FUNCTION_BLOCK Test_DateTimeAsString_ms EXTENDS TUnitTestBase
VAR
END_VAR

METHOD  Execute
VAR_INST
    TimeStruct : TIMESTRUCT := (wDay := 23, wMonth := 12, wYear := 1945, wHour := 22, wMinute := 20, wSecond := 18, wMilliseconds := 512);
END_VAR
Assertion.AssertEquals_STRING(
    Expected := '22:20:18.512 23/12/1945',
    Actual   := F_DateTimeAsString_ms(TimeStruct),
    ObjectName := _TestName,
    VariableName  := 'F_DateTimeAsString_ms(TimeStruct)');


Test_Finished();
END_METHOD

END_FUNCTION_BLOCK

(* stored: Version 1.1.0.1, ProductVersion 3.1.4024.3
   POU Test_DateTimeAsString_ms: Id {e1762af4-84bd-4bfa-ad92-86f0b2f3caa5}, SpecialFunc None
   Method Execute: Id {79e5e476-6795-4fa2-a45a-8bc959bdbcb2} *)
